_CFC_ (* Continuous Function Chart, elements in execution order *)
(* TAMBUR *)
(* SU2 *)
(* VITALNYA *)
(* SU1 *)
(* TOPOCHNA KOMORA *)
#0 MACRO Topochna(pin 1 "button 1": sw_topochna1, pin 2 "button 2": 0, pin 3 "button 3": 0, pin 4 "status": topochna2_l, pin 5 "mooveSensor": moove_topochna, pin 6 "duration": lightDuration, pin 7 "KNX": eib_topochna_l)
	#1 XOR(pin 1, pin 2, pin 3)
	#2 AND(#1, NOT pin 4)
	#3 OR(#2, NOT pin 5, pin 7)
	#4 OR(NOT pin 7, #5)
	#5 AND(#1, pin 4)
	#6 fbTopochna:FB_StairwellLight(#3, #4, #8, t#0ms, t#0ms)
	out 1 "output" <= #6
	#7 MUL(pin 6, msecMultiplier)
	#8 DINT_TO_TIME(#7)
	#9 SUB(#8, fbTopochna.TimerLightDuration.ET)
	out 2 "timeLeft" <= #9
END_MACRO
#10 eib_topochna_l <= #0.out 1
#11 topochna2_l <= #0.out 1
#12 topochna_l <= #0.out 1
#13 fbKomora1_sw:FB_ShortLongClick(sw_komora1, longPressDelay)
#14 MACRO Komora(pin 1 "button 1": #13.out 1, pin 2 "button 2": 0, pin 3 "button 3": sw_topochna2, pin 4 "status": komora_l, pin 5 "mooveSensor": moove_komora, pin 6 "duration": lightDuration, pin 7 "KNX": eib_komora_l)
	#15 XOR(pin 1, pin 2, pin 3)
	#16 AND(#15, NOT pin 4)
	#17 OR(#16, NOT pin 5, pin 7)
	#18 OR(NOT pin 7, #19)
	#19 AND(#15, pin 4)
	#20 fbKomora_l:FB_StairwellLight(#17, #18, #22, t#0ms, t#0ms)
	out 1 "output" <= #20
	#21 MUL(pin 6, msecMultiplier)
	#22 DINT_TO_TIME(#21)
	#23 SUB(#22, fbKomora_l.TimerLightDuration.ET)
	out 2 "timeLeft" <= #23
END_MACRO
#24 eib_komora_l <= #14.out 1
#25 komora_l <= #14.out 1
#26 fbKomoraVent:FB_Light(eib_vent_komora, NOT eib_vent_komora, #13.out 2)
#27 eib_vent_komora <= #26
#28 vent_komora <= #26
#29 fbSu1_1sw:FB_ShortLongClick(sw_su1_1, longPressDelay)
#30 XOR(sw_tambur_su, #29.out 1)
#31 fbSu1_l:FB_Light(eib_su1_l, NOT eib_su1_l, #30)
#32 eib_su1_l <= #31
#33 su1_l <= #31
#34 fbSu1Vent:FB_Light(eib_vent_su1, NOT eib_vent_su1, #29.out 2)
#35 eib_vent_su1 <= #34
#36 vent_su1 <= #34
#37 fbSu1_rakovyna:FB_Light(eib_su1_rakovyna, NOT eib_su1_rakovyna, sw_su1_2)
#38 eib_su1_rakovyna <= #37
#39 su1_rakovyna <= #37
#40 eib_su2_l <= #45
#41 fbSu2_l:FB_Light(eib_su2_l, NOT eib_su2_l, sw_kuh_su2)
#42 eib_su2_l <= #41
#43 su2_l <= #41
#44 fbKuh_su2_sw:FB_ShortLongClick(sw_kuh_su2, longPressDelay)
#45 fbSu2_l:FB_Light(eib_su2_l, NOT eib_su2_l, #44.out 1)
#46 su2_l <= #45
#47 su2_bra <= #93
#48 fbSu2_dush:FB_Light(eib_su2_dush, NOT eib_su2_dush, #44.out 2)
#49 su2_dush <= #48
#50 su2_polytsi <= #48
#51 fbDush_sw:FB_ShortLongClick(sw_su2, longPressDelay)
#52 eib_dush <= #54
#53 eib_su2_bra <= #93
#54 fbDush:FB_Light(eib_dush, NOT eib_dush, #51.out 1)
#55 dush <= #54
#56 eib_vent_dush <= #58
#57 eib_su2_dush <= #48
#58 fbDush_vent:FB_Light(eib_vent_dush, NOT eib_vent_dush, #51.out 2)
#59 vent_dush <= #58
#60 eib_vent_kuh_low <= #66
#61 fbKuh1_sw:FB_ShortLongClick(sw_kuh1, longPressDelay)
#62 fbKuhnya:FB_Light(eib_kuhnya1, NOT eib_kuhnya1, #61.out 1)
#63 kuhnya1 <= #62
#64 eib_kuhnya1 <= #62
#65 kuhnya2 <= #62
#66 fbKuhnyaVent:FB_Light(eib_vent_kuh_low, NOT eib_vent_kuh_low, #61.out 2)
#67 vent_kuh_low <= #66
#68 eib_vitalnya_smugy1 <= #70
#69 XOR(sw_vitalnya1, sw_kuh2)
#70 fbSmugy:FB_Light(eib_vitalnya_smugy1, NOT eib_vitalnya_smugy1, #69)
#71 vitalnya_smugy1 <= #70
#72 vitalnya_smugy2 <= #70
#73 eib_vitalnya_l <= #75
#74 XOR(sw_vitalnya2, sw_kuh4)
#75 fbVitalnya_l:FB_Light(eib_vitalnya_l, NOT eib_vitalnya_l, #74)
#76 vitalnya_l <= #75
#77 fbProkladka:FB_Light(eib_vitalnya_prokladka, NOT eib_vitalnya_prokladka, sw_kuh3)
#78 vitalnya_prokladka <= #77
#79 eib_vitalnya_prokladka <= #77
#80 fbTerassa:FB_Light(eib_terassa, NOT eib_terassa, sw_vitalnya3)
#81 eib_terassa <= #80
#82 terassa <= #80
#83 eib_pidval_shody <= #88
#84 fbSkhody2Pov:FB_Light(eib_skhody2pov, NOT eib_skhody2pov, sw_tambur1_2)
#85 skhody2pov <= #84
#86 eib_skhody2pov <= #84
#87 fbTambur3_sw:FB_ShortLongClick(sw_tambur3, longPressDelay)
#88 fbPidval_shody:FB_Light(eib_pidval_shody, NOT eib_pidval_shody, #87.out 1)
#89 pidval_shody <= #88
#90 AND(bDarkOutside, NOT moove_korydor)
#91 eib_tambur_l <= #97.out 1
#92 tambur_l <= #97.out 1
#93 fbSu2_bra:FB_Light(eib_su2_bra, NOT eib_su2_bra, -)
#94 fbTerassa_stina:FB_Light(eib_terassa_stina, NOT eib_terassa_stina, sw_vitalnya3)
#95 terassa_stina <= #94
#96 eib_terassa_stina <= #94
#97 MACRO Tambur(pin 1 "button 1": sw_tambur1, pin 2 "button 2": sw_vhid1, pin 3 "button 3": 0, pin 4 "status": tambur_l, pin 5 "mooveSensor": #90, pin 6 "duration": lightDuration, pin 7 "KNX": eib_tambur_l)
	#98 XOR(pin 1, pin 2, pin 3)
	#99 AND(#98, NOT pin 4)
	#100 OR(#99, NOT pin 5, pin 7)
	#101 OR(NOT pin 7, #102)
	#102 AND(#98, pin 4)
	#103 fbTamburFirstFloor:FB_StairwellLight(#100, #101, #105, t#0ms, t#0ms)
	out 1 "output" <= #103
	#104 MUL(pin 6, msecMultiplier)
	#105 DINT_TO_TIME(#104)
	#106 SUB(#105, fbTamburFirstFloor.TimerLightDuration.ET)
	out 2 "timeLeft" <= #106
END_MACRO
_END_CFC_
END_PROGRAM
